// Mitsubishi GX Works2 project: 0402_test1   PLC: Q03UDV

PROGRAM MAIN
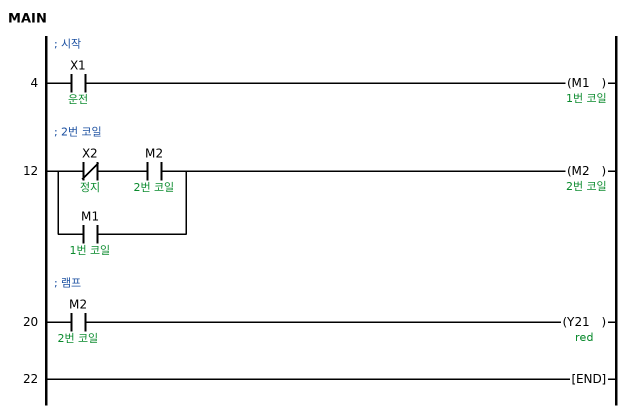
; 시작
4     LD      X1  ; 운전
      OUT     M1  ; 1번 코일
; 2번 코일
12    LDI     X2  ; 정지
      AND     M2  ; 2번 코일
      OR      M1  ; 1번 코일
      OUT     M2  ; 2번 코일
; 램프
20    LD      M2  ; 2번 코일
      OUT     Y21  ; red
22    END
END_PROGRAM
